(* IEC 61131-3 sources: generating_plc_code_with_llms/Code#1/CodeLlama/second run, 17 files *)

(* ---- 10.st ---- *)
// 16.803051948547363s
// 2 (VAR_END fehlt, input variable falsch, RETURN falsch)
```c
FUNCTION SIGMOID(x:REAL):REAL;
VAR
    y:REAL;
BEGIN
    IF x < -50 THEN
        y := 0;
    ELSIF x > 50 THEN
        y := 1;
    ELSE
        y := 1 / (1 + EXP(-x));
    END_IF;
    RETURN y;
END_FUNCTION;
```

(* ---- 11.st ---- *)
// 12.408095121383667s
// 2 (VAR_END fehlt, input variable falsch, RETURN falsch)
```c
FUNCTION SIGN(x:REAL):INTEGER;
VAR
    y:INTEGER;
BEGIN
    IF x > 0 THEN
        y := 1;
    ELSE
        y := -1;
    END_IF;
    RETURN y;
END_FUNCTION;
```

(* ---- 2.st ---- *)
// 22.132529497146606s
// 2 (RETURN falsch)
```c
FUNCTION COEF(N,K):BINOMIAL_COEFFICIENT
VAR
    I:UINT;
    J:UINT;
    RESULT:UINT;
END_VAR
RESULT := 1;
FOR I:=1 TO N DO
    FOR J:=1 TO K DO
        IF (J<=I) THEN
            RESULT := RESULT * (I-J+1)/J;
        END_IF;
    END_FOR;
END_FOR;
RETURN RESULT;
END_FUNCTION
```

(* ---- 21.st ---- *)
// 102.11876630783081s
// 3
```
FUNCTION BURNER : BOOL;
VAR
    PRE_HEAT : BOOL;
    OIL_TEMP : BOOL;
    STAGE2 : BOOL;
    RST : BOOL;
    IN : BOOL;
    FAIL : BOOL;
    STATUS : UINT;
END_VAR
IF (IN = FALSE) THEN
    PRE_HEAT := FALSE;
    OIL_TEMP := FALSE;
    STAGE2 := FALSE;
    RST := FALSE;
    FAIL := FALSE;
    STATUS := 110;
END_IF;
IF (IN = TRUE) THEN
    IF (PRE_HEAT = FALSE) THEN
        PRE_HEAT := TRUE;
        OIL_TEMP := FALSE;
        STAGE2 := FALSE;
        RST := FALSE;
        FAIL := FALSE;
        STATUS := 111;
    END_IF;
    IF (PRE_HEAT = TRUE) THEN
        IF (OIL_TEMP = FALSE) THEN
            OIL_TEMP := TRUE;
            STAGE2 := FALSE;
            RST := FALSE;
            FAIL := FALSE;
            STATUS := 112;
        END_IF;
        IF (OIL_TEMP = TRUE) THEN
            IF (STAGE2 = FALSE) THEN
                STAGE2 := TRUE;
                RST := FALSE;
                FAIL := FALSE;
                STATUS := 113;
            END_IF;
            IF (STAGE2 = TRUE) THEN
                IF (RST = FALSE) THEN
                    RST := TRUE;
                    FAIL := FALSE;
                    STATUS := 110;
                END_IF;
                IF (RST = TRUE) THEN
                    IF (FAIL = FALSE) THEN
                        FAIL := TRUE;
                        STATUS := 9;
                    END_IF;
                    IF (FAIL = TRUE) THEN
                        FAIL := FALSE;
                        STATUS := 110;
                    END_IF;
                END_IF;
            END_IF;
        END_IF;
    END_IF;
END_IF;
BURNER := (PRE_HEAT AND OIL_TEMP) OR STAGE2;
```

(* ---- 14.st ---- *)
// 43.04270315170288s
// 2 (Variablen falsch deklariert)
```
FUNCTION_BLOCK FC1001
VAR
    // Inputs
    INPUT ENABLE : BOOL;
    INPUT SENSOR_VALUE : REAL;
    INPUT SWITCHING_VALUE : REAL;
    INPUT HYSTERESIS : REAL;
    // Outputs
    OUTPUT OUTPUT : BOOL;
END_VAR
IF ENABLE THEN
    IF SENSOR_VALUE > (SWITCHING_VALUE + (HYSTERESIS / 100) * SWITCHING_VALUE) THEN
        OUTPUT := TRUE;
    ELSIF SENSOR_VALUE < (SWITCHING_VALUE - (HYSTERESIS / 100) * SWITCHING_VALUE) THEN
        OUTPUT := FALSE;
    ELSE
        OUTPUT := OUTPUT;
    END_IF;
END_IF;
```

(* ---- 15.st ---- *)
// 32.49787092208862s
// 3 (macht nicht alles was es soll)
```
FUNCTION_BLOCK FC1002
VAR
    P_HU : BOOL;
    P_AL : BOOL;
    E_A : BOOL;
    P1 : BOOL;
END_VAR
IF E_A THEN
    IF NOT P1 THEN
        P1 := TRUE;
        P_HU := FALSE;
        P_AL := FALSE;
    END_IF;
ELSE
    IF P1 THEN
        P1 := FALSE;
        P_HU := FALSE;
        P_AL := FALSE;
    END_IF;
END_IF;
END_FUNCTION_BLOCK
```

(* ---- 18.st ---- *)
// 84.38465976715088s
// 4
```
FUNCTION_BLOCK FC1003
VAR_INPUT
    IN : REAL; (* input value from temperature sensor *)
    IN_MIN : REAL := 0.0; (* lower limit of original range *)
    IN_MAX : REAL := 255.0; (* upper limit of original range *)
    OUT_MIN : REAL := -20.0; (* lower limit of output range *)
    OUT_MAX : REAL := 40.0; (* upper limit of output range *)
END_VAR
VAR_OUTPUT
    OUT : REAL; (* output value for temperature *)
END_VAR
VAR
    RANGE_IN : REAL := IN_MAX - IN_MIN; (* range of original input values *)
    RANGE_OUT : REAL := OUT_MAX - OUT_MIN; (* range of output values *)
    FACTOR : REAL := RANGE_OUT / RANGE_IN; (* factor for scaling *)
END_VAR
IF IN < IN_MIN THEN
    OUT := OUT_MIN;
ELSIF IN > IN_MAX THEN
    OUT := OUT_MAX;
ELSE
    OUT := (IN - IN_MIN) * FACTOR + OUT_MIN;
END_IF;
END_FUNCTION_BLOCK
```

(* ---- 19.st ---- *)
// 63.44924306869507s
// 2 (S1 nicht definiert)
```
FUNCTION_BLOCK FB_1005
VAR_INPUT
START : BOOL;
V_MAX : REAL;
V_MIN : REAL;
END_VAR
VAR_OUTPUT
D_MAX : REAL;
D_MIN : REAL;
END_VAR
VAR
M_MAX : REAL;
M_MIN : REAL;
P1 : BOOL;
END_VAR
IF START THEN
  M_MAX := 0.0;
  M_MIN := 0.0;
  P1 := FALSE;
END_IF
IF NOT(START) AND (M_MAX > V_MAX OR M_MIN < V_MIN) THEN
  P1 := TRUE;
END_IF
IF S1 THEN
  IF M_MAX > M_MIN THEN
    D_MAX := M_MAX;
    D_MIN := M_MIN;
  ELSE
    D_MAX := M_MIN;
    D_MIN := M_MAX;
  END_IF
END_IF
```

(* ---- 3.st ---- *)
// 17.258148193359375s
// 4
```c
FUNCTION_BLOCK Fibonacci
VAR_INPUT
    n : UINT;
END_VAR
VAR_OUTPUT
    f : UINT;
END_VAR
f := 0;
IF n = 1 THEN
    f := 1;
ELSIF n > 1 THEN
    f := Fibonacci(n - 1) + Fibonacci(n - 2);
END_IF;
```

(* ---- 9.st ---- *)
// 19.88591504096985s
// 4
```c
FUNCTION_BLOCK PLC_PROGRAM
VAR_INPUT
    YEAR : INT;
END_VAR
VAR_OUTPUT
    LEAPYEAR : BOOL;
END_VAR
IF (YEAR MOD 4 = 0) AND ((YEAR MOD 100 <> 0) OR (YEAR MOD 400 = 0)) THEN
    LEAPYEAR := TRUE;
ELSE
    LEAPYEAR := FALSE;
END_IF
```

(* ---- 1.st ---- *)
// 22.272629976272583s
// 3
```
PROGRAM AlarmExample
VAR
    xAlarm1 : BOOL;
    xAlarm2 : BOOL;
    xAllOn  : BOOL;
    xAllOff : BOOL;
END_VAR

IF (xAllOn) THEN
    xAlarm1 := TRUE;
    xAlarm2 := TRUE;
ELSIF (xAllOff) THEN
    xAlarm1 := FALSE;
    xAlarm2 := FALSE;
END_IF
```

(* ---- 16.st ---- *)
// 42.21020460128784s
// 2 (Timer nicht richtig ausgelesen)
```
PROGRAM TRAFFIC_LIGHTS;
VAR
	North_green, North_yellow, North_red : BOOL;
	East_green, East_yellow, East_red : BOOL;
	TON : TIME;
END_VAR;

IF TON < 5000 THEN
	North_green := TRUE;
	East_red := TRUE;
ELSIF TON >= 5000 AND TON < 6000 THEN
	North_yellow := TRUE;
	East_red := FALSE;
ELSIF TON >= 9500 AND TON < 10000 THEN
	North_red := TRUE;
	East_green := TRUE;
ELSE
	North_red := FALSE;
	East_yellow := TRUE;
END_IF;
```

(* ---- 20.st ---- *)
// 26.03848958015442s
// 2 (Timer nicht richtig deklariert/initialisiert)
```
PROGRAM Interlock_Example;
VAR
  I1, I2 : BOOL;
  Q1, Q2 : BOOL;
  TL : TIME := 50ms;
END_VAR;

IF (I1 AND NOT(Q1)) OR (I2 AND NOT(Q2)) THEN
  IF (I1 AND NOT(Q1)) THEN
    Q1 := TRUE;
    Q2 := FALSE;
  ELSE
    Q2 := TRUE;
    Q1 := FALSE;
  END_IF;
END_IF;
```

(* ---- 4.st ---- *)
// 24.310040950775146s
// 2
```
PROGRAM fill_level_check;
VAR
    analog_value : WORD;
    percentage : REAL;
    low, ok, high : BOOL;
END_VAR;

CASE percentage OF
    0..10 : low := TRUE;
    11..90 : ok := TRUE;
    91..100 : high := TRUE;
END_CASE;

IF analog_value < 1 THEN
    warning_horn := TRUE;
END_IF;
```

(* ---- 5.st ---- *)
// 38.23284649848938s
// 3
```
PROGRAM GATE_CONTROLLER
VAR
	Start_Loop : BOOL;
	One_Hour_Timer : TON;
	Auth : STRING[10];
	my_defined_str : STRING := '123456789';
END_VAR

IF Start_Loop THEN
	One_Hour_Timer(IN:=TRUE, PT:=T#1h);
ELSE
	IF One_Hour_Timer.Q THEN
		IF Auth = my_defined_str THEN
			Start_Loop := TRUE;
		END_IF
		One_Hour_Timer(IN:=FALSE, PT:=T#1h);
	ELSE
		IF NOT One_Hour_Timer.Q AND Start_Loop THEN
			Start_Loop := FALSE;
		END_IF
	END_IF
END_IF
```

(* ---- 6.st ---- *)
// 63.66718077659607s
// 3
```
PROGRAM CraneLift
VAR
	doConvTop : BOOL;
	doConvBottom : BOOL;
	diConvTop : BOOL;
	diConvBottom : BOOL;
	doLiftTop : BOOL;
	doLiftBottom : BOOL;
	diLiftTop : BOOL;
	diLiftBottom : BOOL;
	doConvLift : BOOL;
	diBoxLift : BOOL;
	doLiftUnload : BOOL;
END_VAR

IF doConvTop THEN
	IF NOT diConvTop THEN
		doLiftTop := TRUE;
	END_IF;
END_IF;

IF doConvBottom THEN
	IF NOT diConvBottom THEN
		doLiftBottom := TRUE;
	END_IF;
END_IF;

IF doLiftTop OR doLiftBottom THEN
	IF NOT (diLiftTop AND diLiftBottom) THEN
		doConvLift := TRUE;
	END_IF;
END_IF;

IF doConvLift THEN
	IF diBoxLift THEN
		doLiftUnload := TRUE;
	END_IF;
END_IF;

IF doLiftUnload THEN
	doConvLift := FALSE;
END_IF;
```

(* ---- 7.st ---- *)
// 32.626829624176025s
// 2 (i ist nicht definiert)
```
PROGRAM Crane;
VAR
  LoadReceptors : ARRAY [1..5] OF INTEGER := (0, 0, 0, 0, 0);
  TotalLoad : INTEGER;
  AverageValue : REAL;
END_VAR;

FOR i := 1 TO 5 DO
  LoadReceptors[i] := AnalogInput(i);
END_FOR;

TotalLoad := 0;
FOR i := 1 TO 5 DO
  TotalLoad := TotalLoad + LoadReceptors[i];
END_FOR;
AverageValue := TotalLoad / 5.0;
```
